// TwinCAT 3 PLC project Untitled1
// ProgramVersion: 3.1.4024.0
// libraries:
//   Tc2_Standard, * (Beckhoff Automation GmbH)
//   Tc2_System, * (Beckhoff Automation GmbH)
//   Tc3_Module, * (Beckhoff Automation GmbH)
//   VisuDialogs, * (System)
//   VisuSymbols,3.5.10.0,System
// project tree:
//   / GlobalTextList.TcGTLO, PlcTask.TcTTO, Task_4.TcTTO, Task_5.TcTTO, Task_6.TcTTO, Task_7.TcTTO
//   GVLs/ GVL.TcGVL
//   POUs/ Programma_4.TcPOU, Programma_2.TcPOU, Programma_test.TcPOU, Programma_1.TcPOU, Programma_3.TcPOU
//   VISUs/ Visualization.TcVIS, VisualizationManager.TcVMO (not stored)
// real-time tasks:
//   TASK PlcTask: cycle T#10ms, priority 20, ADS port 350
//   TASK Task 4: cycle T#10ms, priority 1, ADS port 351
//   TASK Task 5: cycle T#10ms, priority 2, ADS port 352
//   TASK Task 6: cycle T#10ms, priority 3, ADS port 353
//   TASK Task 7: cycle T#10ms, priority 4, ADS port 354

CONFIGURATION Untitled1
    RESOURCE PLC ON TwinCAT3
        TASK PlcTask(INTERVAL := T#10ms, PRIORITY := 20);
        TASK Task_4(INTERVAL := T#10ms, PRIORITY := 1);
        TASK Task_5(INTERVAL := T#10ms, PRIORITY := 2);
        TASK Task_6(INTERVAL := T#10ms, PRIORITY := 3);
        TASK Task_7(INTERVAL := T#10ms, PRIORITY := 4);
        PROGRAM Programma_test WITH PlcTask : Programma_test;
        PROGRAM Programma_1 WITH Task_4 : Programma_1;
        PROGRAM Programma_2 WITH Task_5 : Programma_2;
        PROGRAM Programma_3 WITH Task_6 : Programma_3;
        PROGRAM Programma_4 WITH Task_7 : Programma_4;
    END_RESOURCE
END_CONFIGURATION

// ---- GVLs/GVL.TcGVL
VAR_GLOBAL
    Begin_Knop: BOOL;           // Startknop voor het spel
    Reset_Knop: BOOL;           // Resetknop voor het spel
    Player_1_Lamp: BOOL;        // Lamp voor speler 1 (driehoek)
    Player_2_Lamp: BOOL;        // Lamp voor speler 2 (rondje)
    Player_1: BOOL;             // Is speler 1 aan de beurt?
    Player_2: BOOL;             // Is speler 2 aan de beurt?

    // Rechthoeken voor het bord (9 vakjes)
    Rechthoek_1: BOOL;          // Vak 1
    Rechthoek_2: BOOL;          // Vak 2
    Rechthoek_3: BOOL;          // Vak 3
    Rechthoek_4: BOOL;          // Vak 4
    Rechthoek_5: BOOL;          // Vak 5
    Rechthoek_6: BOOL;          // Vak 6
    Rechthoek_7: BOOL;          // Vak 7
    Rechthoek_8: BOOL;          // Vak 8
    Rechthoek_9: BOOL;          // Vak 9

    // Figuur in elk vak
    Driehoek_1: BOOL;           // Driehoek in vak 1
    Driehoek_2: BOOL;           // Driehoek in vak 2
    Driehoek_3: BOOL;           // Driehoek in vak 3
    Driehoek_4: BOOL;           // Driehoek in vak 4
    Driehoek_5: BOOL;           // Driehoek in vak 5
    Driehoek_6: BOOL;           // Driehoek in vak 6
    Driehoek_7: BOOL;           // Driehoek in vak 7
    Driehoek_8: BOOL;           // Driehoek in vak 8
    Driehoek_9: BOOL;           // Driehoek in vak 9
    Rondje_1: BOOL;             // Rondje in vak 1
    Rondje_2: BOOL;             // Rondje in vak 2
    Rondje_3: BOOL;             // Rondje in vak 3
    Rondje_4: BOOL;             // Rondje in vak 4
    Rondje_5: BOOL;             // Rondje in vak 5
    Rondje_6: BOOL;             // Rondje in vak 6
    Rondje_7: BOOL;             // Rondje in vak 7
    Rondje_8: BOOL;             // Rondje in vak 8
    Rondje_9: BOOL;             // Rondje in vak 9

    // Winconditie en status
    winnaar: INT;               // 0 = geen winnaar, 1 = speler 1, 2 = speler 2
    turn: INT := 0;             // Beurt: 0 = Speler 1, 1 = Speler 2
    game_status: INT := 0;      // Game status: 0 = gestart, 1 = bezig, 2 = gewonnen, 3 = gelijkspel
    selectedSquare: INT := -1;  // Huidige geselecteerde vak
    randomCounter: INT := 0;    // Voor willekeurige speler
END_VAR

// ---- POUs/Programma_test.TcPOU
PROGRAM Programma_test
VAR
END_VAR

END_PROGRAM

// ---- POUs/Programma_1.TcPOU
PROGRAM Programma_1
VAR
	tempRand: INT;  // Tijdelijke variabele voor willekeurige speler
END_VAR

// task 1: 
// Start het spel
IF GVL.game_status = 0 THEN
    IF GVL.Begin_Knop THEN
        // Verhoog de randomCounter voor een willekeurige keuze
        GVL.randomCounter := GVL.randomCounter + 1;
        
        // Genereer een pseudo-willekeurig getal door de randomCounter te delen door 2
        tempRand := GVL.randomCounter MOD 2;  // Dit geeft 0 of 1
        
        IF tempRand = 0 THEN
            GVL.Player_1 := TRUE;
            GVL.Player_2 := FALSE;
            GVL.Player_1_Lamp := TRUE;  // Speler 1 Lamp aan
            GVL.Player_2_Lamp := FALSE;
        ELSE
            GVL.Player_1 := FALSE;
            GVL.Player_2 := TRUE;
            GVL.Player_1_Lamp := FALSE;
            GVL.Player_2_Lamp := TRUE;  // Speler 2 Lamp aan
        END_IF
        GVL.game_status := 1;  // Zet het spel in de "bezig" status
    END_IF
END_IF

END_PROGRAM

// ---- POUs/Programma_2.TcPOU
PROGRAM Programma_2
VAR
    currentPlayer: BOOL;  // Bepaalt welke speler aan de beurt is
	zetGedaan: BOOL;
END_VAR

// task 2: 
// Speler zet zijn figuur
IF GVL.game_status = 1 THEN
    zetGedaan := FALSE; // Variabele om bij te houden of er een zet is gedaan

    // Bepaal welke speler aan de beurt is
    IF GVL.Player_1 THEN
        currentPlayer := TRUE;   // Speler 1 is actief
    ELSE
        currentPlayer := FALSE;  // Speler 2 is actief
    END_IF

    // Controleer of een rechthoek is geselecteerd en of deze leeg is
    // Als de rechthoek leeg is, vul het met het figuur van de speler
    IF GVL.Rechthoek_1 AND NOT (GVL.Driehoek_1 OR GVL.Rondje_1) THEN
        IF currentPlayer THEN
            GVL.Driehoek_1 := TRUE;  // Zet driehoek van speler 1
        ELSE
            GVL.Rondje_1 := TRUE;    // Zet rondje van speler 2
        END_IF
        zetGedaan := TRUE;
    ELSIF GVL.Rechthoek_2 AND NOT (GVL.Driehoek_2 OR GVL.Rondje_2) THEN
        IF currentPlayer THEN
            GVL.Driehoek_2 := TRUE;  // Zet driehoek van speler 1
        ELSE
            GVL.Rondje_2 := TRUE;    // Zet rondje van speler 2
        END_IF
        zetGedaan := TRUE;
    ELSIF GVL.Rechthoek_3 AND NOT (GVL.Driehoek_3 OR GVL.Rondje_3) THEN
        IF currentPlayer THEN
            GVL.Driehoek_3 := TRUE;  // Zet driehoek van speler 1
        ELSE
            GVL.Rondje_3 := TRUE;    // Zet rondje van speler 2
        END_IF
        zetGedaan := TRUE;
    ELSIF GVL.Rechthoek_4 AND NOT (GVL.Driehoek_4 OR GVL.Rondje_4) THEN
        IF currentPlayer THEN
            GVL.Driehoek_4 := TRUE;  // Zet driehoek van speler 1
        ELSE
            GVL.Rondje_4 := TRUE;    // Zet rondje van speler 2
        END_IF
        zetGedaan := TRUE;
    ELSIF GVL.Rechthoek_5 AND NOT (GVL.Driehoek_5 OR GVL.Rondje_5) THEN
        IF currentPlayer THEN
            GVL.Driehoek_5 := TRUE;  // Zet driehoek van speler 1
        ELSE
            GVL.Rondje_5 := TRUE;    // Zet rondje van speler 2
        END_IF
        zetGedaan := TRUE;
    ELSIF GVL.Rechthoek_6 AND NOT (GVL.Driehoek_6 OR GVL.Rondje_6) THEN
        IF currentPlayer THEN
            GVL.Driehoek_6 := TRUE;  // Zet driehoek van speler 1
        ELSE
            GVL.Rondje_6 := TRUE;    // Zet rondje van speler 2
        END_IF
        zetGedaan := TRUE;
    ELSIF GVL.Rechthoek_7 AND NOT (GVL.Driehoek_7 OR GVL.Rondje_7) THEN
        IF currentPlayer THEN
            GVL.Driehoek_7 := TRUE;  // Zet driehoek van speler 1
        ELSE
            GVL.Rondje_7 := TRUE;    // Zet rondje van speler 2
        END_IF
        zetGedaan := TRUE;
    ELSIF GVL.Rechthoek_8 AND NOT (GVL.Driehoek_8 OR GVL.Rondje_8) THEN
        IF currentPlayer THEN
            GVL.Driehoek_8 := TRUE;  // Zet driehoek van speler 1
        ELSE
            GVL.Rondje_8 := TRUE;    // Zet rondje van speler 2
        END_IF
        zetGedaan := TRUE;
    ELSIF GVL.Rechthoek_9 AND NOT (GVL.Driehoek_9 OR GVL.Rondje_9) THEN
        IF currentPlayer THEN
            GVL.Driehoek_9 := TRUE;  // Zet driehoek van speler 1
        ELSE
            GVL.Rondje_9 := TRUE;    // Zet rondje van speler 2
        END_IF
        zetGedaan := TRUE;
    END_IF

    // Wissel de beurt alleen als er een zet is gedaan
    IF zetGedaan THEN
        IF GVL.Player_1 THEN
            GVL.Player_1 := FALSE;   // Zet speler 1 uit
            GVL.Player_2 := TRUE;    // Zet speler 2 aan
            GVL.Player_1_Lamp := FALSE;  // Zet lamp van speler 1 uit
            GVL.Player_2_Lamp := TRUE;   // Zet lamp van speler 2 aan
        ELSE
            GVL.Player_1 := TRUE;    // Zet speler 1 aan
            GVL.Player_2 := FALSE;   // Zet speler 2 uit
            GVL.Player_1_Lamp := TRUE;  // Zet lamp van speler 1 aan
            GVL.Player_2_Lamp := FALSE;  // Zet lamp van speler 2 uit
        END_IF

        // Zet de status van het spel naar 2 (wincheck fase) als er een zet is gedaan
        GVL.game_status := 2;  // Ga naar de wincheck fase
    END_IF
END_IF

END_PROGRAM

// ---- POUs/Programma_3.TcPOU
PROGRAM Programma_3
VAR
    winCondition: BOOL;
END_VAR

// task 3: 
IF GVL.game_status = 2 THEN  // Wincheck fase
    // Controleer of er een winnaar is
    IF (GVL.Driehoek_1 AND GVL.Driehoek_2 AND GVL.Driehoek_3) OR
       (GVL.Driehoek_4 AND GVL.Driehoek_5 AND GVL.Driehoek_6) OR
       (GVL.Driehoek_7 AND GVL.Driehoek_8 AND GVL.Driehoek_9) OR
       (GVL.Driehoek_1 AND GVL.Driehoek_4 AND GVL.Driehoek_7) OR
       (GVL.Driehoek_2 AND GVL.Driehoek_5 AND GVL.Driehoek_8) OR
       (GVL.Driehoek_3 AND GVL.Driehoek_6 AND GVL.Driehoek_9) OR
       (GVL.Driehoek_1 AND GVL.Driehoek_5 AND GVL.Driehoek_9) OR
       (GVL.Driehoek_3 AND GVL.Driehoek_5 AND GVL.Driehoek_7) THEN
        // Speler 1 heeft gewonnen
        GVL.winnaar := 1;
        GVL.Player_1_Lamp := TRUE;
        GVL.game_status := 3;  // Zet status naar "gewonnen"
        
    ELSIF (GVL.Rondje_1 AND GVL.Rondje_2 AND GVL.Rondje_3) OR
           (GVL.Rondje_4 AND GVL.Rondje_5 AND GVL.Rondje_6) OR
           (GVL.Rondje_7 AND GVL.Rondje_8 AND GVL.Rondje_9) OR
           (GVL.Rondje_1 AND GVL.Rondje_4 AND GVL.Rondje_7) OR
           (GVL.Rondje_2 AND GVL.Rondje_5 AND GVL.Rondje_8) OR
           (GVL.Rondje_3 AND GVL.Rondje_6 AND GVL.Rondje_9) OR
           (GVL.Rondje_1 AND GVL.Rondje_5 AND GVL.Rondje_9) OR
           (GVL.Rondje_3 AND GVL.Rondje_5 AND GVL.Rondje_7) THEN
        // Speler 2 heeft gewonnen
        GVL.winnaar := 2;
        GVL.Player_2_Lamp := TRUE;
        GVL.game_status := 3;  // Zet status naar "gewonnen"
        
    ELSE
        // Als er geen winnaar is, controleer dan of het gelijkspel is
        IF (GVL.Driehoek_1 OR GVL.Rondje_1) AND
           (GVL.Driehoek_2 OR GVL.Rondje_2) AND
           (GVL.Driehoek_3 OR GVL.Rondje_3) AND
           (GVL.Driehoek_4 OR GVL.Rondje_4) AND
           (GVL.Driehoek_5 OR GVL.Rondje_5) AND
           (GVL.Driehoek_6 OR GVL.Rondje_6) AND
           (GVL.Driehoek_7 OR GVL.Rondje_7) AND
           (GVL.Driehoek_8 OR GVL.Rondje_8) AND
           (GVL.Driehoek_9 OR GVL.Rondje_9) THEN
            // Het is gelijkspel
            GVL.game_status := 4;  // Zet status naar gelijkspel
        ELSE
            // Er zijn nog lege vakken, geen gelijkspel
            GVL.game_status := 1;  // Ga terug naar de beurtfase
        END_IF
    END_IF
END_IF

END_PROGRAM

// ---- POUs/Programma_4.TcPOU
PROGRAM Programma_4
VAR
END_VAR

//task 4: 
// Reset alle variabelen naar de beginstatus
IF GVL.Reset_Knop THEN
    // Reset alle variabelen
    GVL.Driehoek_1 := FALSE; GVL.Driehoek_2 := FALSE; GVL.Driehoek_3 := FALSE;
    GVL.Driehoek_4 := FALSE; GVL.Driehoek_5 := FALSE; GVL.Driehoek_6 := FALSE;
    GVL.Driehoek_7 := FALSE; GVL.Driehoek_8 := FALSE; GVL.Driehoek_9 := FALSE;
    GVL.Rondje_1 := FALSE; GVL.Rondje_2 := FALSE; GVL.Rondje_3 := FALSE;
    GVL.Rondje_4 := FALSE; GVL.Rondje_5 := FALSE; GVL.Rondje_6 := FALSE;
    GVL.Rondje_7 := FALSE; GVL.Rondje_8 := FALSE; GVL.Rondje_9 := FALSE;

    GVL.Player_1_Lamp := FALSE; GVL.Player_2_Lamp := FALSE;
    GVL.Player_1 := FALSE; GVL.Player_2 := FALSE;
    GVL.winnaar := 0; GVL.game_status := 0; GVL.turn := 0;
END_IF

END_PROGRAM

// ---- GlobalTextList.TcGTLO
TEXTLIST GlobalTextList
  209 = 'Begin'
  562 = 'BEGIN'
  618 = 'Gellijkspel'
  350 = 'Gewonnen'
  608 = 'Player 1'
  677 = 'Player 2'
  337 = 'RESEt'
  419 = 'RESET'
END_TEXTLIST

// ---- VISUs/Visualization.TcVIS
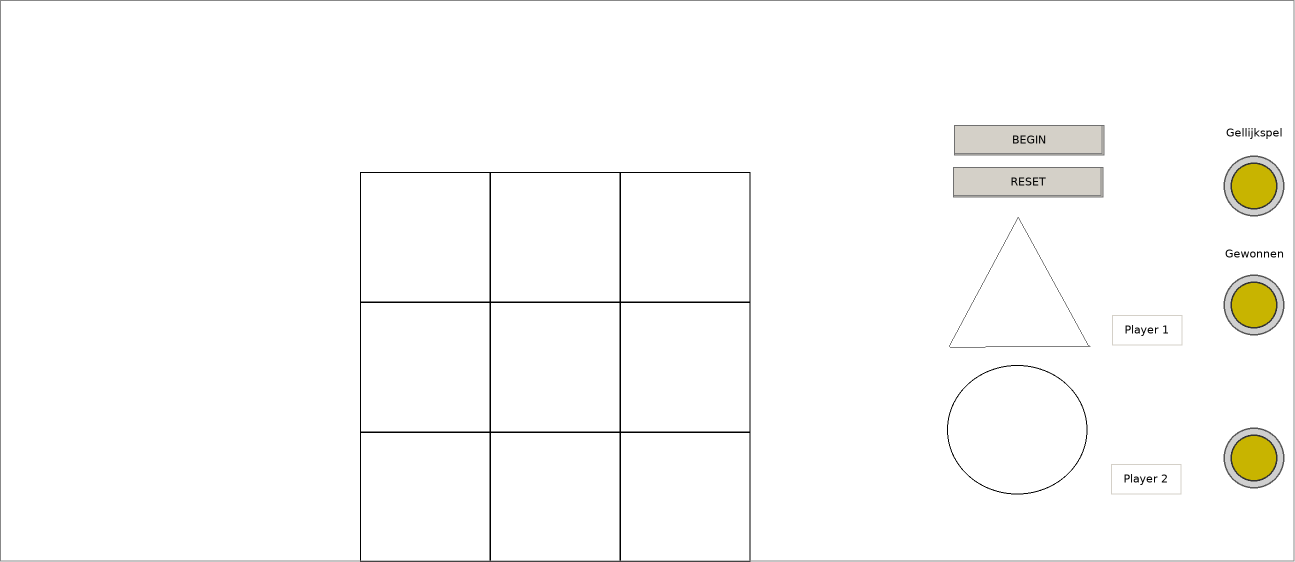
VISUALIZATION Visualization  // 1295x562
    Rectangle (360,172 130x130)
        tap GVL.Rechthoek_1
    Rectangle (490,172 130x130)
        tap GVL.Rechthoek_2
    Rectangle (620,172 130x130)
        tap GVL.Rechthoek_3
    Rectangle (360,302 130x130)
        tap GVL.Rechthoek_4
    Rectangle (490,302 130x130)
        tap GVL.Rechthoek_5
    Rectangle (620,302 130x130)
        tap GVL.Rechthoek_6
    Rectangle (360,432 130x130)
        tap GVL.Rechthoek_7
    Rectangle (490,432 130x130)
        tap GVL.Rechthoek_8
    Rectangle (620,432 130x130)
        tap GVL.Rechthoek_9
    Textfield (1112,315 70x30), "Player 1"
    Textfield (1111,464 70x30), "Player 2"
    Button (954,125 150x30), "BEGIN"
        tap GVL.Begin_Knop
    Polygon (949,346) (1018,217) (1088,345) (1090,346) (950,347), colour toggle: GVL.Player_1_Lamp
    Ellipse (947,365 140x129), colour toggle: GVL.Player_2_Lamp
    Button (953,167 150x30), "RESET"
        tap GVL.Reset_Knop
    Ellipse (363,175 125x125), colour toggle: GVL.Rondje_1
        tap GVL.Rechthoek_1
    Ellipse (493,175 125x125), colour toggle: GVL.Rondje_2
        tap GVL.Rechthoek_2
    Ellipse (623,175 125x125), colour toggle: GVL.Rondje_3
        tap GVL.Rechthoek_3
    Ellipse (623,305 125x125), colour toggle: GVL.Rondje_6
        tap GVL.Rechthoek_6
    Ellipse (493,305 125x125), colour toggle: GVL.Rondje_5
        tap GVL.Rechthoek_5
    Ellipse (363,305 125x125), colour toggle: GVL.Rondje_4
        tap GVL.Rechthoek_4
    Ellipse (363,435 125x125), colour toggle: GVL.Rondje_7
        tap GVL.Rechthoek_7
    Ellipse (493,435 125x125), colour toggle: GVL.Rondje_8
        tap GVL.Rechthoek_8
    Ellipse (623,435 125x125), colour toggle: GVL.Rondje_9
        tap GVL.Rechthoek_9
    Polygon (363,297) (428,177) (488,297) (488,297) (363,297), colour toggle: GVL.Driehoek_1
        tap GVL.Rechthoek_1
    Polygon (493,297) (558,177) (618,297) (618,297) (493,297), colour toggle: GVL.Driehoek_2
        tap GVL.Rechthoek_2
    Polygon (623,297) (688,177) (748,297) (748,297) (623,297), colour toggle: GVL.Driehoek_3
        tap GVL.Rechthoek_3
    Polygon (623,427) (688,307) (748,427) (748,427) (623,427), colour toggle: GVL.Driehoek_6
        tap GVL.Rechthoek_6
    Polygon (493,427) (558,307) (618,427) (618,427) (493,427), colour toggle: GVL.Driehoek_5
        tap GVL.Rechthoek_5
    Polygon (363,427) (428,307) (488,427) (488,427) (363,427), colour toggle: GVL.Driehoek_4
        tap GVL.Rechthoek_4
    Polygon (623,557) (688,437) (748,557) (748,557) (623,557), colour toggle: GVL.Driehoek_9
        tap GVL.Rechthoek_9
    Polygon (493,557) (558,437) (618,557) (618,557) (493,557), colour toggle: GVL.Driehoek_8
        tap GVL.Rechthoek_8
    Polygon (363,557) (428,437) (488,557) (488,557) (363,557), colour toggle: GVL.Driehoek_7
        tap GVL.Rechthoek_7
    Lamp1 (1219,270 70x70), variable: Player_1_Lamp_G, style: Lamp-Lamp1-Yellow
    Lamp1 (1219,423 70x70), variable: Player_2_Lamp_G, style: Lamp-Lamp1-Yellow
    Label (1214,239 81x30), "Gewonnen"
    Lamp1 (1219,151 70x70), variable: Gelijkspel, style: Lamp-Lamp1-Yellow
    Label (1214,118 81x30), "Gellijkspel"
END_VISUALIZATION
